TYPE TxHmi :
STRUCT
	t : REAL := 0.0;
	em1500 : TxHmiStewart;
	em8000 : TxHmiStewart;
	comau : TxHmiComau;
	at960 : TxHmiLeica;	
	mru1 : TxHmiMru;
	mru2 : TxHmiMru;
END_STRUCT
END_TYPE

(* stored: Version 1.1.0.1, ProductVersion 3.1.4020.12
   DUT TxHmi: Id {2cfd4700-2b83-4fe6-81fa-843b179f6b37} *)
